KUKA KRL program: Makrosaw.src

&ACCESS RV
&PARAM TEMPLATE = C:\KRC\Roboter\Template\makrosawvorgabe.src
&PARAM EDITMASK = MakroSAW
&PARAM TPVW_VERSION=8.3.18
DEF  MAKROSAW ( )
; FOLD Makro Anfang;%{PSE} %MKUKATPVW
SPS_N=-1
; ENDFOLD
; FOLD ;%{H}
END
; ENDFOLD
